{attribute 'hide_all_locals'}
FUNCTION_BLOCK PUBLIC FB_FullTimeEmployee_2 EXTENDS FB_Employee_1
VAR_INPUT
END_VAR
VAR_OUTPUT
END_VAR
VAR
	nAnnualSalaryBacking	:	UINT;
END_VAR

METHOD PUBLIC GetMonthlySalary : LREAL
VAR_INPUT
END_VAR
GetMonthlySalary := nAnnualSalary / 12;
END_METHOD

{attribute 'monitoring' := 'variable'}
PROPERTY PUBLIC nAnnualSalary : UINT
GET
nAnnualSalary := nAnnualSalaryBacking;
END_GET
SET
nAnnualSalaryBacking := nAnnualSalary;
END_SET
END_PROPERTY

END_FUNCTION_BLOCK

(* stored: Version 1.1.0.1, ProductVersion 3.1.4024.12
   POU FB_FullTimeEmployee_2: Id {d5681875-7aac-49c7-a04d-5ea70283a5eb}, SpecialFunc None
   Method GetMonthlySalary: Id {87fc335a-e0a0-40cb-8af0-62afa113a8aa}
   Property nAnnualSalary: Id {bd569f95-43b4-4924-9fca-c1280c82edf7}
   Get Get: Id {5c12615e-a145-40a0-87fc-90c8c7fa0646}
   Set Set: Id {517538e6-4c3d-48a0-b0c2-0e0b0b6708bc} *)
